(* CODESYS project SysSocket_unix.ecp

Project tree, tasks and I/O mapping:
  Controller : 750-8212 PFC200 2ETH RS, WAGO, order no. 0750-8212, version 5.14.3.54
    application Application
      libraries: ; WagoSysBSDSocket, 1.1.1.0 (WAGO); CmpErrors, 3.3.1.40 (System); WagoSysPlainMem, 1.5.2.0 (WAGO); SysSocket, 3.5.14.0 (System)
      task PLC_Task (cyclic, interval t#50ms, priority 15) calls Client
      program Client [ST]
      data type sockaddr_un
      data type usun_path
      global variables GVL
      program eresult_Errno [ST]
    Kbus : Kbus, WAGO, version 1.4.0.2
        unmapped channels: K-BUS diagnostics
    MODBUS
      MODBUS : MODBUS, WAGO, order no. n/a, version 1.1.1.15
    Common.PCI
    Serial
      COM1 : COM1, WAGO, version 0.0.0.19
*)

// Controller/Application/sockaddr_un


TYPE sockaddr_un :
STRUCT
	sa_family_t : WagoSysBSDSocket.sa_family_t; 
	usun_path : usun_path;  
END_STRUCT
END_TYPE

(*
http://manpages.org/af_unix/7

A UNIX domain socket address is represented in the following
structure:

#define UNIX_PATH_MAX    108
struct sockaddr_un {
    sa_family_t sun_family;               /* AF_UNIX */
    char sun_path[UNIX_PATH_MAX];  /* pathname */
};

***********

From #include <sys/socket.h>

"struct sockaddr" is a generic definition. It's used by any socket function that requires an address.
A struct sockaddr should generally only be used as the base type for a pointer. 
It is a structure intended to cover the common initial sequence of the members in the address family specific socket address types: 
struct sockaddr_un, struct sockaddr_in, struct sockaddr_in6 etc.)

struct sockaddr
  {
    __SOCKADDR_COMMON (sa_);	/* Common data: address family and length.  */
    char sa_data[14];		/* Address data.  */
  };


*)

//http://www.cas.mcmaster.ca/~qiao/courses/cs3mh3/tutorials/socket.html

// Since Unix domain and Internet domain have different address structures as shown earlier, type casting is needed.

// Dette skulle være riktig definisjon av Berkley AF_UNIX socket


(*

Since Unix domain and Internet domain have different address structures as shown earlier, type casting is needed.
                   #define                        SERV_PATH        "./serv.path"
                    struct sockaddr_un serv_addr;
                    int servlen;

                    serv_addr.sun_family = AF_UNIX;
                    strcpy(serv_addr.sun_path, SERV_PATH);
                    servlen = strlen(serv_addr.sun_path) + sizeof(serv)_addr.sun_family); *)
           //        bind(sockfd, (struct sockaddr *) &serv_addr, servlen);  
					
//Note that the BSD network system calls do not assume that the Unix pathname in sun_path is terminated with a null type.  We can initialize the address by:
//                   bzero((char *) &serv_addr, sizeof(serv_addr));
//After the call bind, the system knows the name OF the host socket.  In the Unix domain CASE, it is a path name.

// Controller/Application/usun_path
TYPE usun_path :
UNION
sun_path : 	STRING(gcUNIX_PATH_MAX);
absun_path : ARRAY [1..gcUNIX_PATH_MAX] OF BYTE;  // 1 byte on 32 bit
END_UNION
END_TYPE

// Controller/Application/GVL

VAR_GLOBAL CONSTANT
	
	gcUNIX_PATH_MAX : BYTE := 108; 

END_VAR

// Controller/Application/Client
PROGRAM Client
VAR
	
	// Sys library
	sockfd : SysSocket.SysTypes.RTS_IEC_HANDLE;
	sockaddr : sockaddr_un; 
	// Wago library
	sockfd_wago: WagoSysBSDSocket.sockhandle_t; // Wago socket filedescriptor, alias for RTS_IEC_HANDLE
	socketaddr_wago : WagoSysBSDSocket.unSockaddr;
	RTC_IEC_RESULT: SysSocket.RTS_IEC_RESULT; // For connect
	eResult_wago_create: WagoSysBSDSocket.eResultCode;	
	eResult_wago_connect: WagoSysBSDSocket.eResultCode;
	
	// Test typecast
	soccaddress : syssocket.SOCKADDRESS;
	
	sPath : STRING := 'a';
	iError : INT;
	bTxData : BYTE := 1;
	xCreate: BOOL;
	xCreate_wago : BOOL;
	xSend: BOOL;
	udiLen : UDINT;
	xError : BOOL;
	xConnect : BOOL;
	xConnect_wago : BOOL;
END_VAR


// SysSocket create
IF xCreate THEN
	// Create socket / socket descriptor
	sockfd := SysSocket.SysSockCreate(iAddressFamily:= SysSocket.SOCKET_AF_UNIX, diType:= SysSocket.SOCKET_STREAM, diProtocol:= 0, pResult:= ADR(RTC_IEC_RESULT)); // RTC_IEC_RESULT == 1 ??
	
	IF sockfd <> 0 THEN
		xCreate := FALSE;
	ELSE
		xCreate := FALSE;
		iError := 1;
	END_IF
	
	// Name the socket
	sockaddr.sa_family_t := SysSocket.SOCKET_AF_UNIX; 
	sockaddr.usun_path.sun_path := 'a';
	
END_IF

// WagoSysBSDSocket create
IF xCreate_wago THEN
	// Create socket / socket descriptor (sockhandle_t is ALIAS for RTS_IEC_HANDLE)
	sockfd_wago := WagoSysBSDSocket.FuSock_Socket(eDomain:= WagoSysBSDSocket.AF_LOCAL, eType:= WagoSysBSDSocket.SOCK_STREAM, eProtocol:= 0, eResult=> eResult_wago_create);

	IF sockfd_wago <> 0 THEN
		xCreate_wago := FALSE;
	ELSE
		xCreate_wago := FALSE;
		iError := 2;
	END_IF
	
	// Har Wago riktig struktur ????
	//socketaddr_wago.sa_family := WagoSysBSDSocket.AF_LOCAL;
	//socketaddr_wago.in := ??
	
	// Name the socket - bruker egen
	sockaddr.sa_family_t := WagoSysBSDSocket.AF_LOCAL; 
	sockaddr.usun_path.sun_path := 'a';

END_IF


// Open virker ikke
// mulig må typecast riktig ???  connect(client_sock, (struct sockaddr *) &server_sockaddr, len);

// Connect by SysSocket
IF xConnect THEN
	udiLen := WagoAppString.Length(sTr:= sockaddr.usun_path.sun_path) + SIZEOF(sockaddr.sa_family_t); // servlen = strlen(serv_addr.sun_path) + sizeof(serv_addr.sun_family); // 1 (a) + 2 (AF_UNIX)
	RTC_IEC_RESULT := SysSocket.SysSockConnect(hSocket:= sockfd, pSockAddr:= ADR(sockaddr.usun_path.sun_path), diSockAddrSize:= UDINT_TO_DINT(udiLen)); // 209
	xConnect := FALSE;	
END_IF

// Connect by WagoSysBSDSocket
IF xConnect_wago THEN
	udiLen := WagoAppString.Length(sTr:= sockaddr.usun_path.sun_path) + SIZEOF(sockaddr.sa_family_t); // servlen = strlen(serv_addr.sun_path) + sizeof(serv_addr.sun_family); // 1 (a) + 2 (AF_UNIX)
	xError := WagoSysBSDSocket.FuSock_Connect(Socket:= sockfd_wago, pAddress:= ADR(sockaddr), udiAddress_len:= udiLen, eResult=> eResult_wago_connect); // 135 - Unspecified
	
	IF eResult_wago_connect = 0 AND NOT xError THEN
		xConnect_wago := FALSE;
	ELSE
		xConnect_wago := FALSE;
		iError := 4;
	END_IF
	
END_IF	
	

(*
IF xSend THEN
	// Send data
	SysSocket.SysSockSend(
		hSocket:= sockfd, 
		pbyBuffer:= ADR(bTxData), 
		diBufferSize:= SIZEOF(bTxData), 
		diFlags:= 0, 
		pResult:= ADR(RTC_IEC_RESULT));
	
		IF RTC_IEC_RESULT <> 0 THEN
			iError := 2;	
		ELSE
			xSend := FALSE;
		END_IF
		
		
END_IF

*)

END_PROGRAM

// Controller/Application/eresult_Errno
PROGRAM eresult_Errno
VAR
END_VAR


(*

e!cockpit

ERRORS:

In case of success this function returns 0 (FALSE) and the output eResult shows 0=OK. In case of failure, the return value is TRUE and the output eResult indicates the error cause as described below.

The FuSock_Connect() function will fail if:

ENOTSOCK (mandatory for POSIX compliance): The Socket argument is was either not generated by this library, or was deallocated already or does not qualify to be a proper socket by other reasons. 
ECONNREFUSED (mandatory for POSIX compliance): The target address was not listening for connections or refused the connection request. 
EINPROGRESS (mandatory for POSIX compliance): O_NONBLOCK is set for the socket handle for the socket and the connection cannot be immediately established; the connection will be established asynchronously. 
EUNSPECIFIC: A general problem with this function is encountered and no further details about the reason are available. (none known so far) 
ENOSUCCESS: An unexpected problem with this function is encountered with a differenciated reason that does not does not fit into the POSIX scheme. 
The FuSock_Connect() function may fail if:

EADDRNOTAVAIL (mandatory for POSIX compliance): The specified address is not available from the local machine. 
EAFNOSUPPORT (mandatory for POSIX compliance): The specified address is not a valid address for the address family of the specified socket. 
EISCONN (mandatory for POSIX compliance): The specified socket is connection-mode and is already connected. 
EBADF (mandatory for POSIX compliance): The socket argument is not a valid socket handle. 
ETIMEDOUT (mandatory for POSIX compliance): The attempt to connect timed out before a connection was made. 
EALREADY (mandatory for POSIX compliance): A connection request is already in progress for the specified socket. 
EPROTOTYPE (mandatory for POSIX compliance): The specified address has a different type than the socket bound to the specified peer address. 
EHOSTUNREACH (optional): The destination host cannot be reached (probably because the host is down or a remote router cannot reach it). 
EINVAL (optional): The address_len argument is not a valid length for the address family; or invalid address family in the sockaddr structure. 
EADDRINUSE (optional): Attempt to establish a connection that uses addresses that are already in use. 
ENOBUFS (optional): No buffer space is available. 
The FuSock_Connect() function may also fail in future releases if:

ENETUNREACH (mandatory for POSIX compliance): No route to the network is present. (actual firmware does not differentiate between ENETUNREACH and EHOSTUNREACH.) 
EACCES (optional): Search permission is denied for a component of the path prefix; or write access to the named socket is denied. 
ECONNRESET (optional): Remote host reset the connection request. 
ELOOP (optional): Too many symbolic links were encountered during resolution of the pathname in address. 
ENAMETOOLONG (optional): The length of a pathname is too long. 
ENETDOWN (optional): The local network interface used to reach the destination is down. 
EOPNOTSUPP (optional): The socket is listening and cannot be connected. 
Deviation from POSIX.1-2008:

The error code is uniformly provided via the additional output variable eResult:eResultCode, which contains the values specified by POSIX. The POSIX constructs errno or getlasterror() are not supported. 
The output is typed as BOOL (not as int), in order to provide the same functionality for Codesys as intended by POSIX for C. 
In certain conditions the system might not be able to deliver differentiated result codes as requested by the POSIX standard. In those cases, where the exact cause cannot be differentiated from other causes, the result codes EUNSPECIFIC and ENOSUCCESS are is returned instead. These codes are not contained in the original POSIX specification. EUNSPECIFIC is used in cases where the system notifies that it cannot differentiate the cause at all (ERR_FAILED), while ENOSUCCESS is used when the result code from the system is somewhat differentiated, but cannot be mapped unambiguously to the POSIX requirements. 
Error EINVAL if pAddress is a null-pointer 





From errno.h


#define	EPERM		 1	/* Operation not permitted */
#define	ENOENT		 2	/* No such file or directory */
#define	ESRCH		 3	/* No such process */
#define	EINTR		 4	/* Interrupted system call */
#define	EIO		 5	/* I/O error */
#define	ENXIO		 6	/* No such device or address */
#define	E2BIG		 7	/* Argument list too long */
#define	ENOEXEC		 8	/* Exec format error */
#define	EBADF		 9	/* Bad file number */
#define	ECHILD		10	/* No child processes */
#define	EAGAIN		11	/* Try again */
#define	ENOMEM		12	/* Out of memory */
#define	EACCES		13	/* Permission denied */
#define	EFAULT		14	/* Bad address */
#define	ENOTBLK		15	/* Block device required */
#define	EBUSY		16	/* Device or resource busy */
#define	EEXIST		17	/* File exists */
#define	EXDEV		18	/* Cross-device link */
#define	ENODEV		19	/* No such device */
#define	ENOTDIR		20	/* Not a directory */
#define	EISDIR		21	/* Is a directory */
#define	EINVAL		22	/* Invalid argument */
#define	ENFILE		23	/* File table overflow */
#define	EMFILE		24	/* Too many open files */
#define	ENOTTY		25	/* Not a typewriter */
#define	ETXTBSY		26	/* Text file busy */
#define	EFBIG		27	/* File too large */
#define	ENOSPC		28	/* No space left on device */
#define	ESPIPE		29	/* Illegal seek */
#define	EROFS		30	/* Read-only file system */
#define	EMLINK		31	/* Too many links */
#define	EPIPE		32	/* Broken pipe */
#define	EDOM		33	/* Math argument out of domain of func */
#define	ERANGE		34	/* Math result not representable */

#define	EDEADLK		35	/* Resource deadlock would occur */
#define	ENAMETOOLONG	36	/* File name too long */
#define	ENOLCK		37	/* No record locks available */

/*
 * This error code is special: arch syscall entry code will return
 * -ENOSYS if users try to call a syscall that doesn't exist.  To keep
 * failures of syscalls that really do exist distinguishable from
 * failures due to attempts to use a nonexistent syscall, syscall
 * implementations should refrain from returning -ENOSYS.
 */
#define	ENOSYS		38	/* Invalid system call number */

#define	ENOTEMPTY	39	/* Directory not empty */
#define	ELOOP		40	/* Too many symbolic links encountered */
#define	EWOULDBLOCK	EAGAIN	/* Operation would block */
#define	ENOMSG		42	/* No message of desired type */
#define	EIDRM		43	/* Identifier removed */
#define	ECHRNG		44	/* Channel number out of range */
#define	EL2NSYNC	45	/* Level 2 not synchronized */
#define	EL3HLT		46	/* Level 3 halted */
#define	EL3RST		47	/* Level 3 reset */
#define	ELNRNG		48	/* Link number out of range */
#define	EUNATCH		49	/* Protocol driver not attached */
#define	ENOCSI		50	/* No CSI structure available */
#define	EL2HLT		51	/* Level 2 halted */
#define	EBADE		52	/* Invalid exchange */
#define	EBADR		53	/* Invalid request descriptor */
#define	EXFULL		54	/* Exchange full */
#define	ENOANO		55	/* No anode */
#define	EBADRQC		56	/* Invalid request code */
#define	EBADSLT		57	/* Invalid slot */

#define	EDEADLOCK	EDEADLK

#define	EBFONT		59	/* Bad font file format */
#define	ENOSTR		60	/* Device not a stream */
#define	ENODATA		61	/* No data available */
#define	ETIME		62	/* Timer expired */
#define	ENOSR		63	/* Out of streams resources */
#define	ENONET		64	/* Machine is not on the network */
#define	ENOPKG		65	/* Package not installed */
#define	EREMOTE		66	/* Object is remote */
#define	ENOLINK		67	/* Link has been severed */
#define	EADV		68	/* Advertise error */
#define	ESRMNT		69	/* Srmount error */
#define	ECOMM		70	/* Communication error on send */
#define	EPROTO		71	/* Protocol error */
#define	EMULTIHOP	72	/* Multihop attempted */
#define	EDOTDOT		73	/* RFS specific error */
#define	EBADMSG		74	/* Not a data message */
#define	EOVERFLOW	75	/* Value too large for defined data type */
#define	ENOTUNIQ	76	/* Name not unique on network */
#define	EBADFD		77	/* File descriptor in bad state */
#define	EREMCHG		78	/* Remote address changed */
#define	ELIBACC		79	/* Can not access a needed shared library */
#define	ELIBBAD		80	/* Accessing a corrupted shared library */
#define	ELIBSCN		81	/* .lib section in a.out corrupted */
#define	ELIBMAX		82	/* Attempting to link in too many shared libraries */
#define	ELIBEXEC	83	/* Cannot exec a shared library directly */
#define	EILSEQ		84	/* Illegal byte sequence */
#define	ERESTART	85	/* Interrupted system call should be restarted */
#define	ESTRPIPE	86	/* Streams pipe error */
#define	EUSERS		87	/* Too many users */
#define	ENOTSOCK	88	/* Socket operation on non-socket */
#define	EDESTADDRREQ	89	/* Destination address required */
#define	EMSGSIZE	90	/* Message too long */
#define	EPROTOTYPE	91	/* Protocol wrong type for socket */
#define	ENOPROTOOPT	92	/* Protocol not available */
#define	EPROTONOSUPPORT	93	/* Protocol not supported */
#define	ESOCKTNOSUPPORT	94	/* Socket type not supported */
#define	EOPNOTSUPP	95	/* Operation not supported on transport endpoint */
#define	EPFNOSUPPORT	96	/* Protocol family not supported */
#define	EAFNOSUPPORT	97	/* Address family not supported by protocol */
#define	EADDRINUSE	98	/* Address already in use */
#define	EADDRNOTAVAIL	99	/* Cannot assign requested address */
#define	ENETDOWN	100	/* Network is down */
#define	ENETUNREACH	101	/* Network is unreachable */
#define	ENETRESET	102	/* Network dropped connection because of reset */
#define	ECONNABORTED	103	/* Software caused connection abort */
#define	ECONNRESET	104	/* Connection reset by peer */
#define	ENOBUFS		105	/* No buffer space available */
#define	EISCONN		106	/* Transport endpoint is already connected */
#define	ENOTCONN	107	/* Transport endpoint is not connected */
#define	ESHUTDOWN	108	/* Cannot send after transport endpoint shutdown */
#define	ETOOMANYREFS	109	/* Too many references: cannot splice */
#define	ETIMEDOUT	110	/* Connection timed out */
#define	ECONNREFUSED	111	/* Connection refused */
#define	EHOSTDOWN	112	/* Host is down */
#define	EHOSTUNREACH	113	/* No route to host */
#define	EALREADY	114	/* Operation already in progress */
#define	EINPROGRESS	115	/* Operation now in progress */
#define	ESTALE		116	/* Stale file handle */
#define	EUCLEAN		117	/* Structure needs cleaning */
#define	ENOTNAM		118	/* Not a XENIX named type file */
#define	ENAVAIL		119	/* No XENIX semaphores available */
#define	EISNAM		120	/* Is a named type file */
#define	EREMOTEIO	121	/* Remote I/O error */
#define	EDQUOT		122	/* Quota exceeded */

#define	ENOMEDIUM	123	/* No medium found */
#define	EMEDIUMTYPE	124	/* Wrong medium type */
#define	ECANCELED	125	/* Operation Canceled */
#define	ENOKEY		126	/* Required key not available */
#define	EKEYEXPIRED	127	/* Key has expired */
#define	EKEYREVOKED	128	/* Key has been revoked */
#define	EKEYREJECTED	129	/* Key was rejected by service */

/* for robust mutexes */
#define	EOWNERDEAD	130	/* Owner died */
#define	ENOTRECOVERABLE	131	/* State not recoverable */

#define ERFKILL		132	/* Operation not possible due to RF-kill */

#define EHWPOISON	133	/* Memory page has hardware error */

*)

END_PROGRAM
